{attribute addProperty BoxType "EK1100-0000-0018"}
{attribute addProperty Id "Beckhoff_ELM31xxEK1122Beckhoff_ELM31xxEK1122_3E17608C162A_0001_ELM3102_0000_0016ELM3102_1C598C2535244A_0002_ELM3102_0000_0017ELM3102_1C598C2535244A_0003_ELM3102_0000_0018ELM3102_1C598C2535244A_0004_ELM3104_0000_0016ELM3104_EF18820948060A_0005_ELM3104_0000_0017ELM3104_EF18820948060A_0006_ELM3104_0000_0018ELM3104_EF18820948060A_0007_ELM3142_0000_0016ELM3142_1C598C2535244A_0008_ELM3142_0000_0017ELM3142_1C598C2535244A_0009_ELM3144_0000_0016ELM3144_EF18820948060A_0010_ELM3144_0000_0017ELM3144_EF18820948060A_0011_ELM3146_0000_0016ELM3146_71F10A1860876A_0012_ELM3146_0000_0017ELM3146_71F10A1860876A_0013_ELM3146_0000_0018ELM3146_71F10A1860876A_0014_ELM3148_0000_0017ELM3148_AE8DF5B573692A_0015_ELM3148_0000_0018ELM3148_AE8DF5B573692A_0016_ELM3148_0000_0019ELM3148_AE8DF5B573692"}
{attribute addProperty CRC "3528593069"}
{attribute addProperty SizeInBites "8208"}
{attribute addProperty SizeInBytes "1026"}
TYPE Beckhoff_ELM31xx_D2520EAD EXTENDS EK1100_179A0949 :
STRUCT
	{attribute addProperty Name "Beckhoff_ELM31xxEK1122"}
	Beckhoff_ELM31xxEK1122 : Beckhoff_ELM31xxEK1122_3E17608C;
	{attribute addProperty Name "A_0001_ELM3102_0000_0016"}
	A_0001_ELM3102_0000_0016 : ELM3102_1C598C25;
	{attribute addProperty Name "A_0002_ELM3102_0000_0017"}
	A_0002_ELM3102_0000_0017 : ELM3102_1C598C25;
	{attribute addProperty Name "A_0003_ELM3102_0000_0018"}
	A_0003_ELM3102_0000_0018 : ELM3102_1C598C25;
	{attribute addProperty Name "A_0004_ELM3104_0000_0016"}
	A_0004_ELM3104_0000_0016 : ELM3104_EF188209;
	{attribute addProperty Name "A_0005_ELM3104_0000_0017"}
	A_0005_ELM3104_0000_0017 : ELM3104_EF188209;
	{attribute addProperty Name "A_0006_ELM3104_0000_0018"}
	A_0006_ELM3104_0000_0018 : ELM3104_EF188209;
	{attribute addProperty Name "A_0007_ELM3142_0000_0016"}
	A_0007_ELM3142_0000_0016 : ELM3142_1C598C25;
	{attribute addProperty Name "A_0008_ELM3142_0000_0017"}
	A_0008_ELM3142_0000_0017 : ELM3142_1C598C25;
	{attribute addProperty Name "A_0009_ELM3144_0000_0016"}
	A_0009_ELM3144_0000_0016 : ELM3144_EF188209;
	{attribute addProperty Name "A_0010_ELM3144_0000_0017"}
	A_0010_ELM3144_0000_0017 : ELM3144_EF188209;
	{attribute addProperty Name "A_0011_ELM3146_0000_0016"}
	A_0011_ELM3146_0000_0016 : ELM3146_71F10A18;
	{attribute addProperty Name "A_0012_ELM3146_0000_0017"}
	A_0012_ELM3146_0000_0017 : ELM3146_71F10A18;
	{attribute addProperty Name "A_0013_ELM3146_0000_0018"}
	A_0013_ELM3146_0000_0018 : ELM3146_71F10A18;
	{attribute addProperty Name "A_0014_ELM3148_0000_0017"}
	A_0014_ELM3148_0000_0017 : ELM3148_AE8DF5B5;
	{attribute addProperty Name "A_0015_ELM3148_0000_0018"}
	A_0015_ELM3148_0000_0018 : ELM3148_AE8DF5B5;
	{attribute addProperty Name "A_0016_ELM3148_0000_0019"}
	A_0016_ELM3148_0000_0019 : ELM3148_AE8DF5B5;
END_STRUCT
END_TYPE

(* stored: Version 1.2.0.0, ProductVersion 3.1.4024.9
   DUT Beckhoff_ELM31xx_D2520EAD: Id {d9cc61df-e81e-4789-8186-64100a1816b8} *)
